RoboDK station: Seguir_Trayectoria_3.rdk

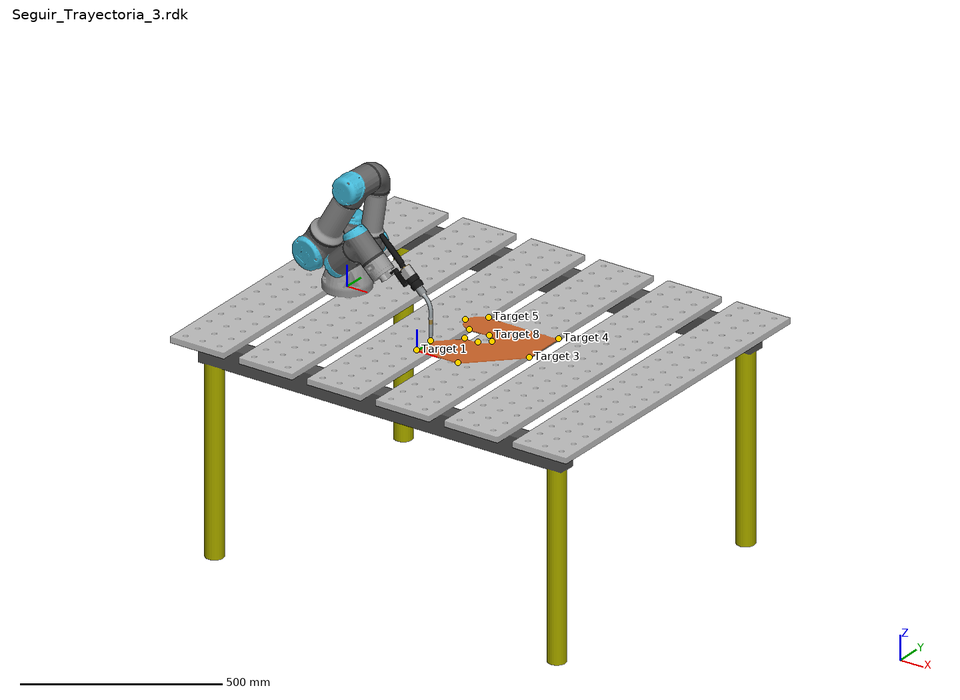
[picture v0: the station drawn from its stored meshes, robots at their saved joint values, targets as dots, program paths as lines]
Station Seguir_Trayectoria_3 (saved by RoboDK 5.7.3). Poses are relative to the parent item; angles as X-Y-Z fixed-axis rotations.
  - frame UR3e Base at (-400, 0, 0) mm
    - robot UR3e: 6 axes, payload 3 kg, reach 500 mm, repeatability 0.03 mm, weight 11 kg
        modified DH rows (alpha deg, a mm, theta deg, d mm): 0, 0, 0, 151.9; 90, 0, 180, 0; 0, 243.55, 0, 0; 0, 213.2, 0, 131.05; -90, 0, 0, 85.35; 90, 0, 180, 92.1
        joint limits [-360, -360, -360, -360, -360, -360] to [360, 360, 360, 360, 360, 360]; home [0, -90, -90, 0, 90, 0]; saved at [-3.341, -120.223, -158.586, 53.76, 92.362, 87.636]
      - tool OTC Daihen FD-84 Welding Gun, TCP at (1, 0, 201) mm, rotated rx 0 ry 45 rz 0 deg, size 100.8 x 32.5 x 283.9 mm
  - object Table 1200x1000mm (Welding) at (0, 0, 0) mm, size 1193.8 x 965.2 x 609.6 mm, geometry from Table-1200x1000mm-Welding.sld
  - frame ref_objeto at (-50, -200, 0) mm
    - object Cutting sheet at (0, 0, 0) mm, size 250 x 250 x 3 mm, geometry from Cutting sheet.STEP
    - target Target 1 (Cartesian target) at (-1, -1, 4) mm, rotated rx 180 ry 0 rz -180 deg; joints [-22.537, -118.8, -143.495, 35.021, 105.725, 73.647] of UR3e
    - target Target 2 (Cartesian target) at (125.4, -1, 4) mm, rotated rx 180 ry 0 rz 180 deg; joints [-13.803, -128.441, -114.677, 17.278, 99.713, 80.145] of UR3e
    - target Target 3 (Cartesian target) at (251, 124.59, 4) mm, rotated rx 180 ry 0 rz -180 deg; joints [8.223, -138.071, -91.678, 4.453, 84.196, 95.834] of UR3e
    - target Target 4 (Cartesian target) at (251, 251.25, 4) mm, rotated rx -180 ry 0 rz -180 deg; joints [26.639, -136.44, -94.121, 2.352, 71.516, 109.529] of UR3e
    - target Target 5 (Cartesian target) at (40, 251.25, 4) mm, rotated rx -180 ry 0 rz 180 deg; joints [59.081, -105.923, -165.286, 28.405, 52.654, 139.734] of UR3e
    - target Target 6 (Cartesian target) at (-1, 210, 4) mm, rotated rx 180 ry 0 rz -180 deg; joints [70.606, -92.827, -186.97, 28.166, 48.165, 153.533] of UR3e
    - target Target 7 (Cartesian target) at (40, 169, 4) mm, rotated rx -180 ry 0 rz -180 deg; joints [35.187, -119.202, -165.149, 53.609, 65.954, 116.499] of UR3e
    - target Target 8 (Cartesian target) at (100, 169, 4) mm, rotated rx 180 ry 0 rz 180 deg; joints [25.018, -118.476, -143.941, 34.599, 72.6, 108.263] of UR3e
    - target Target 9 (Cartesian target) at (124, 145, 4) mm, rotated rx -180 ry 0 rz -180 deg; joints [17.062, -121.33, -134.77, 29.811, 78.026, 102.244] of UR3e
    - target Target 10 (Cartesian target) at (100, 121, 4) mm, rotated rx -180 ry 0 rz -180 deg; joints [12.82, -120.172, -140.014, 34.462, 80.973, 99.141] of UR3e
    - target Target 11 (Cartesian target) at (59.59, 121, 4) mm, rotated rx -180 ry 0 rz -180 deg; joints [15.718, -118.499, -152.481, 44.889, 78.957, 101.254] of UR3e
    - target Target 12 (Cartesian target) at (-1, 60.41, 4) mm, rotated rx 180 ry 0 rz 180 deg; joints [-3.341, -120.223, -158.586, 53.76, 92.362, 87.636] of UR3e
